{attribute addProperty BoxType "EL3182-0000-0016"}
{attribute addProperty Id "Ch_1Ch_1_9A58320E3240Ch_2Ch_2_6B3549513240WcStateAT %I*WcState_F855686C1620InfoDataAT %I*InfoData_275E3363128160"}
{attribute addProperty CRC "2035140665"}
{attribute addProperty SizeInBites "208"}
{attribute addProperty SizeInBytes "26"}
TYPE EL3182_8DBFD1BF :
STRUCT
	{attribute addProperty Name "Ch_1"}
	Ch_1 : Ch_1_9A58320E;
	{attribute addProperty Name "Ch_2"}
	Ch_2 : Ch_2_6B354951;
	{attribute addProperty Name "WcState"}
	WcState : WcState_F855686C;
	{attribute addProperty Name "InfoData"}
	InfoData : InfoData_275E3363;
END_STRUCT
END_TYPE

(* stored: Version 1.2.0.0, ProductVersion 3.1.4024.9
   DUT EL3182_8DBFD1BF: Id {355f26c5-5d27-43cf-9c55-25934b26cd4b} *)
